// TIA Portal V17 export
// export: Created 2023-02-13T11:16:44.7326633Z, ExportSetting WithDefaults, DisplayName Totally Integrated Automation Portal, DisplayVersion V17, DisplayName TIA Portal Openness, DisplayVersion V17, DisplayName TIA Portal Teamcenter Gateway, DisplayVersion V17, DisplayName TIA Portal Version Control Interface, DisplayVersion V17, DisplayName SINAMICS Startdrive Advanced, DisplayVersion V17, DisplayName SINAMICS Startdrive G130, G150, S120, S150, SINAMICS MV, S210, DisplayVersion V17, DisplayName SINAMICS Startdrive G110M, G120, G120C, G120D, G120P, G115D, DisplayVersion V17, DisplayName STEP 7 Professional, DisplayVersion V17, DisplayName STEP 7 Safety, DisplayVersion V17, DisplayName WinCC Professional, DisplayVersion V17
ORGANIZATION_BLOCK "Cyclic interrupt"   // OB30, LAD, CyclicInterrupt
{ S7_Optimized_Access := 'TRUE' }
VERSION : 0.1
// stored: AutoNumber true, IsIECCheckEnabled false, SetENOAutomatically false
   VAR_INPUT
      Initial_Call : Bool;   // Initial call of this OB
      Event_Count : Int;   // Events discarded
   END_VAR
   VAR_TEMP   // added for the SCL form of the ladder/FBD networks
      _w1 : Bool;
      _w2 : Bool;
      _w3 : Bool;
      _w4 : Bool;
      _w5 : Bool;
   END_VAR
BEGIN

REGION Network 1
   // "IO Analog Preparation_DB"."TT-01.01".QOUT
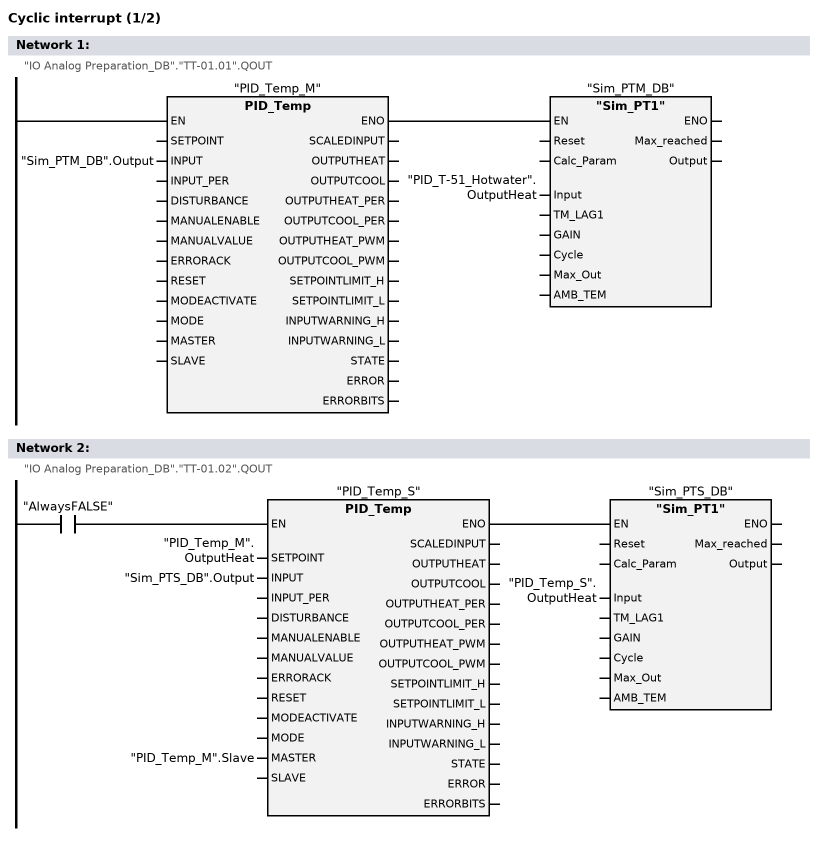
   RUNG wire#powerrail
      "PID_Temp_M".PID_Temp(Setpoint :=, Input := "Sim_PTM_DB".Output, Input_PER :=, Disturbance :=, ManualEnable :=, ManualValue :=, ErrorAck :=, Reset :=, ModeActivate :=, Mode :=, Master :=, Slave :=, ScaledInput =>, OutputHeat =>, OutputCool =>, OutputHeat_PER =>, OutputCool_PER =>, OutputHeat_PWM =>, OutputCool_PWM =>, SetpointLimit_H =>, SetpointLimit_L =>, InputWarning_H =>, InputWarning_L =>, State =>, Error =>, ErrorBits =>)
      "Sim_PTM_DB"(Reset :=, Calc_Param :=, Input := "PID_T-51_Hotwater".OutputHeat, TM_LAG1 :=, GAIN :=, Cycle :=, Max_Out :=, AMB_TEM :=, Max_reached =>, Output =>)
   END_RUNG
   // the same network as SCL:
   "PID_Temp_M"(Input := "Sim_PTM_DB".Output, ENO => #_w1);   // PID_Temp
   IF #_w1 THEN
       "Sim_PTM_DB"(Input := "PID_T-51_Hotwater".OutputHeat);   // "Sim_PT1"
   END_IF;
END_REGION

REGION Network 2
   // "IO Analog Preparation_DB"."TT-01.02".QOUT
   RUNG wire#powerrail
      Contact( "AlwaysFALSE" )
      "PID_Temp_S".PID_Temp(Setpoint := "PID_Temp_M".OutputHeat, Input := "Sim_PTS_DB".Output, Input_PER :=, Disturbance :=, ManualEnable :=, ManualValue :=, ErrorAck :=, Reset :=, ModeActivate :=, Mode :=, Master := "PID_Temp_M".Slave, Slave :=, ScaledInput =>, OutputHeat =>, OutputCool =>, OutputHeat_PER =>, OutputCool_PER =>, OutputHeat_PWM =>, OutputCool_PWM =>, SetpointLimit_H =>, SetpointLimit_L =>, InputWarning_H =>, InputWarning_L =>, State =>, Error =>, ErrorBits =>)
      "Sim_PTS_DB"(Reset :=, Calc_Param :=, Input := "PID_Temp_S".OutputHeat, TM_LAG1 :=, GAIN :=, Cycle :=, Max_Out :=, AMB_TEM :=, Max_reached =>, Output =>)
   END_RUNG
   // the same network as SCL:
   "PID_Temp_S"(EN := "AlwaysFALSE",   // PID_Temp
                Setpoint := "PID_Temp_M".OutputHeat,
                Input := "Sim_PTS_DB".Output,
                Master := "PID_Temp_M".Slave,
                ENO => #_w1);
   IF #_w1 THEN
       "Sim_PTS_DB"(Input := "PID_Temp_S".OutputHeat);   // "Sim_PT1"
   END_IF;
END_REGION

REGION Network 3: PID HotWater T51 Control
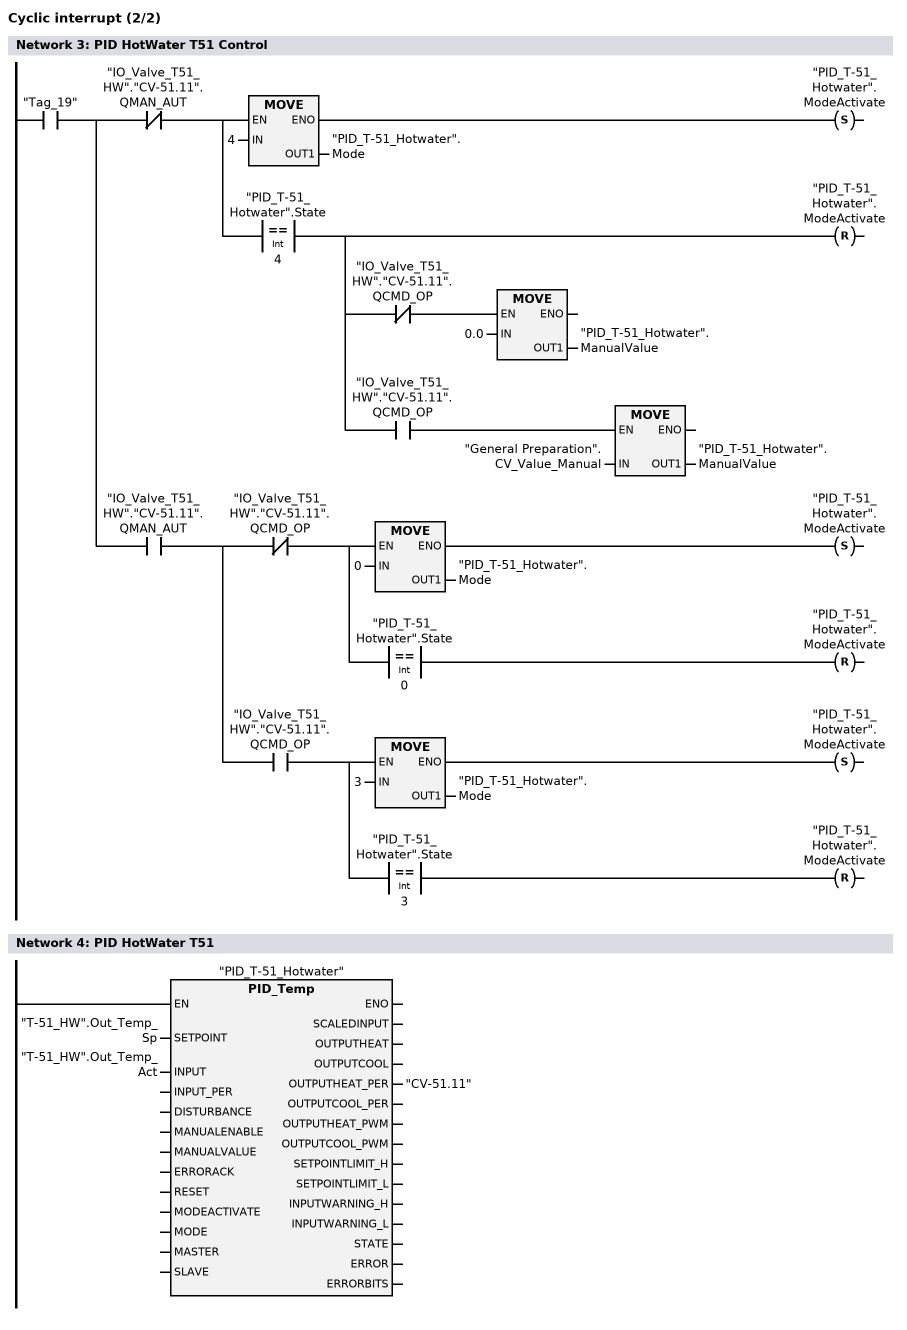
   RUNG wire#powerrail
      Contact( "Tag_19" )
      wire#w1
      I_Contact( "IO_Valve_T51_HW"."CV-51.11".QMAN_AUT )
      wire#w2
      Move(in := 4, out1 => "PID_T-51_Hotwater".Mode)
      S_Coil( "PID_T-51_Hotwater".ModeActivate )
   END_RUNG
   RUNG wire#w2
      { S7_Templates := "SrcType := Int" } EQ_Contact(in1 := "PID_T-51_Hotwater".State, in2 := 4)
      wire#w3
      R_Coil( "PID_T-51_Hotwater".ModeActivate )
   END_RUNG
   RUNG wire#w3
      I_Contact( "IO_Valve_T51_HW"."CV-51.11".QCMD_OP )
      Move(in := 0.0, out1 => "PID_T-51_Hotwater".ManualValue)
   END_RUNG
   RUNG wire#w3
      Contact( "IO_Valve_T51_HW"."CV-51.11".QCMD_OP )
      Move(in := "General Preparation".CV_Value_Manual, out1 => "PID_T-51_Hotwater".ManualValue)
   END_RUNG
   RUNG wire#w1
      Contact( "IO_Valve_T51_HW"."CV-51.11".QMAN_AUT )
      wire#w4
      I_Contact( "IO_Valve_T51_HW"."CV-51.11".QCMD_OP )
      wire#w5
      Move(in := 0, out1 => "PID_T-51_Hotwater".Mode)
      S_Coil( "PID_T-51_Hotwater".ModeActivate )
   END_RUNG
   RUNG wire#w5
      { S7_Templates := "SrcType := Int" } EQ_Contact(in1 := "PID_T-51_Hotwater".State, in2 := 0)
      R_Coil( "PID_T-51_Hotwater".ModeActivate )
   END_RUNG
   RUNG wire#w4
      Contact( "IO_Valve_T51_HW"."CV-51.11".QCMD_OP )
      wire#w6
      Move(in := 3, out1 => "PID_T-51_Hotwater".Mode)
      S_Coil( "PID_T-51_Hotwater".ModeActivate )
   END_RUNG
   RUNG wire#w6
      { S7_Templates := "SrcType := Int" } EQ_Contact(in1 := "PID_T-51_Hotwater".State, in2 := 3)
      R_Coil( "PID_T-51_Hotwater".ModeActivate )
   END_RUNG
   // the same network as SCL:
   #_w1 := "Tag_19" AND NOT "IO_Valve_T51_HW"."CV-51.11".QMAN_AUT;
   IF #_w1 THEN
       "PID_T-51_Hotwater".Mode := 4;
       "PID_T-51_Hotwater".ModeActivate := TRUE;
   END_IF;
   #_w2 := #_w1 AND ("PID_T-51_Hotwater".State = 4);
   IF #_w2 THEN "PID_T-51_Hotwater".ModeActivate := FALSE; END_IF;
   IF #_w2 AND NOT "IO_Valve_T51_HW"."CV-51.11".QCMD_OP THEN "PID_T-51_Hotwater".ManualValue := 0.0; END_IF;
   IF #_w2 AND "IO_Valve_T51_HW"."CV-51.11".QCMD_OP THEN
       "PID_T-51_Hotwater".ManualValue := "General Preparation".CV_Value_Manual;
   END_IF;
   #_w3 := "Tag_19" AND "IO_Valve_T51_HW"."CV-51.11".QMAN_AUT;
   #_w4 := #_w3 AND NOT "IO_Valve_T51_HW"."CV-51.11".QCMD_OP;
   IF #_w4 THEN
       "PID_T-51_Hotwater".Mode := 0;
       "PID_T-51_Hotwater".ModeActivate := TRUE;
   END_IF;
   IF #_w4 AND ("PID_T-51_Hotwater".State = 0) THEN "PID_T-51_Hotwater".ModeActivate := FALSE; END_IF;
   #_w5 := #_w3 AND "IO_Valve_T51_HW"."CV-51.11".QCMD_OP;
   IF #_w5 THEN
       "PID_T-51_Hotwater".Mode := 3;
       "PID_T-51_Hotwater".ModeActivate := TRUE;
   END_IF;
   IF #_w5 AND ("PID_T-51_Hotwater".State = 3) THEN "PID_T-51_Hotwater".ModeActivate := FALSE; END_IF;
END_REGION

REGION Network 4: PID HotWater T51
   RUNG wire#powerrail
      "PID_T-51_Hotwater".PID_Temp(Setpoint := "T-51_HW".Out_Temp_Sp, Input := "T-51_HW".Out_Temp_Act, Input_PER :=, Disturbance :=, ManualEnable :=, ManualValue :=, ErrorAck :=, Reset :=, ModeActivate :=, Mode :=, Master :=, Slave :=, ScaledInput =>, OutputHeat =>, OutputCool =>, OutputHeat_PER => "CV-51.11", OutputCool_PER =>, OutputHeat_PWM =>, OutputCool_PWM =>, SetpointLimit_H =>, SetpointLimit_L =>, InputWarning_H =>, InputWarning_L =>, State =>, Error =>, ErrorBits =>)
   END_RUNG
   // the same network as SCL:
   "PID_T-51_Hotwater"(Setpoint := "T-51_HW".Out_Temp_Sp,   // PID_Temp
                       Input := "T-51_HW".Out_Temp_Act,
                       OutputHeat_PER => "CV-51.11");
END_REGION
END_ORGANIZATION_BLOCK
